TYPE E_HMIstatus :
(
	Off := 0,
	Standby,
	On,
	Autotune,
	IdleLoad
);
END_TYPE

(* stored: Version 1.1.0.1, ProductVersion 3.1.0.26
   DUT E_HMIstatus: Id {b481d7d9-95f8-4f85-8d05-02a0b9c78214} *)
